// Mitsubishi GX Works2 project: 21_01   PLC: FX3G

// global labels: Global1
VAR_GLOBAL
  switch_check_start AT X007 : BOOL;
  finish_packing AT Y002 : BOOL;
  Not_sufficnt_stuff AT M1 : BOOL;
  kashut_container AT D1101 : REAL;
  lata_container AT D1201 : REAL;
  shmarim_container AT D1202 : REAL;
END_VAR
VAR_GLOBAL CONSTANT
  con120 : REAL := 120;
  cons6 : REAL := 6;
  cons54 : REAL := 54;
END_VAR
VAR_GLOBAL
  Y_7 AT Y007 : BOOL;
  X_11 AT X011 : BOOL;
  Urgent_Shut AT X011 : BOOL;
  start_cook AT X001 : BOOL;
  analog_input AT D8281 : INT;
END_VAR
VAR_GLOBAL CONSTANT
  con400 : INT := 400;
END_VAR
VAR_GLOBAL
  correct_analog AT D1111 : INT;
END_VAR
VAR_GLOBAL CONSTANT
  cons_5 : INT := 5;
END_VAR
VAR_GLOBAL
  what_is_it AT M12 : BOOL;
  NO AT M12 : BOOL;
  Yes_Lager AT M12 : BOOL;
END_VAR
VAR_GLOBAL CONSTANT
  cons_120 : REAL := 120;
  cons_6 : REAL := 6;
END_VAR
VAR_GLOBAL
  bishul_container AT D1299 : REAL;
END_VAR
VAR_GLOBAL CONSTANT
  cons_54 : REAL := 54;
  cons_150 : REAL := 150;
  cons_12 : REAL := 12;
  cons_60 : REAL := 60;
END_VAR
VAR_GLOBAL
  Y_3 AT Y003 : BOOL;
  M_12 AT M12 : BOOL;
  M_13 AT M13 : BOOL;
  Yes_philenzer AT M12 : BOOL;
END_VAR
VAR_GLOBAL CONSTANT
  cons_0 : REAL;
  cons_126 : REAL := 126;
END_VAR
VAR_GLOBAL
  M_17 AT M17 : BOOL;
  cooke_timer AT TC5 : BOOL;
END_VAR
VAR_GLOBAL CONSTANT
  sec_4 : INT := 40;
END_VAR
VAR_GLOBAL
  stop_cooke AT TS5 : BOOL;
  stop_cook AT TS5 : BOOL;
  lamp1_off AT Y001 : BOOL;
  X_5 AT X005 : BOOL;
  tsisa_container AT D1301 : REAL;
  end_cook_lam AT M3 : BOOL;
  BE_counter AT TC2 : BOOL;
END_VAR
VAR_GLOBAL CONSTANT
  Four_sec : INT := 40;
END_VAR
VAR_GLOBAL
  BE_OFF AT TS2 : BOOL;
  Helo_Lamp AT M0 : BOOL;
  Timer_1 AT TC3 : BOOL;
END_VAR
VAR_GLOBAL CONSTANT
  One_sec : INT := 10;
END_VAR
VAR_GLOBAL
  end_timer1 AT TS3 : BOOL;
  Lamp_1 AT Y004 : BOOL;
  Lamp_4 AT Y004 : BOOL;
  Timer_2 AT TC4 : BOOL;
  end_Timer2 AT TS4 : BOOL;
  lamp3 AT Y003 : BOOL;
  lamp0 AT Y003 : BOOL;
  lamlam AT X003 : BOOL;
END_VAR
VAR_GLOBAL CONSTANT
  cons0 : REAL;
END_VAR
VAR_GLOBAL
  BD_counter AT TC6 : BOOL;
  BD_OFF AT TS6 : BOOL;
END_VAR
VAR_GLOBAL CONSTANT
  Three_sec : INT := 30;
END_VAR
VAR_GLOBAL
  Timer_3 AT TC7 : BOOL;
  end_timer3 AT TS7 : BOOL;
  Timer_4 AT TC8 : BOOL;
  end_Timer4 AT TS8 : BOOL;
  Helo_Lamp2 AT M2 : BOOL;
  start_pac AT X002 : BOOL;
  end_tsisa AT M5 : BOOL;
  Nora AT Y006 : BOOL;
  cc1_counter AT CC1 : BOOL;
END_VAR
VAR_GLOBAL CONSTANT
  count1 : WORD := K1;
END_VAR
VAR_GLOBAL
  cc6_counter AT CC6 : BOOL;
END_VAR
VAR_GLOBAL CONSTANT
  count6 : WORD := K6;
END_VAR
VAR_GLOBAL
  cs1 AT CS1 : BOOL;
  cs6 AT CS6 : BOOL;
  y_2 AT Y002 : BOOL;
  x_0 AT X000 : BOOL;
  ready_container AT D1401 : REAL;
END_VAR
VAR_GLOBAL CONSTANT
  add_abeer : REAL := 6;
  add_shishia : REAL := 1;
  con_40 : REAL := 40;
END_VAR
VAR_GLOBAL
  D_4001 AT D4001 : REAL;
  analog_output AT D8282 : INT;
  D_4000 AT D4000 : REAL;
  break AT M14 : BOOL;
END_VAR
VAR_GLOBAL CONSTANT
  mul_1 : REAL := 1;
END_VAR

// task Task_01 (event TRUE, interval 0, priority 31): POU_01

PROGRAM POU_01
(* structured ladder/FBD written out as ST: instructions are called as NAME(EN, inputs, outputs); _pN, _eN, _tN stand for wires *)
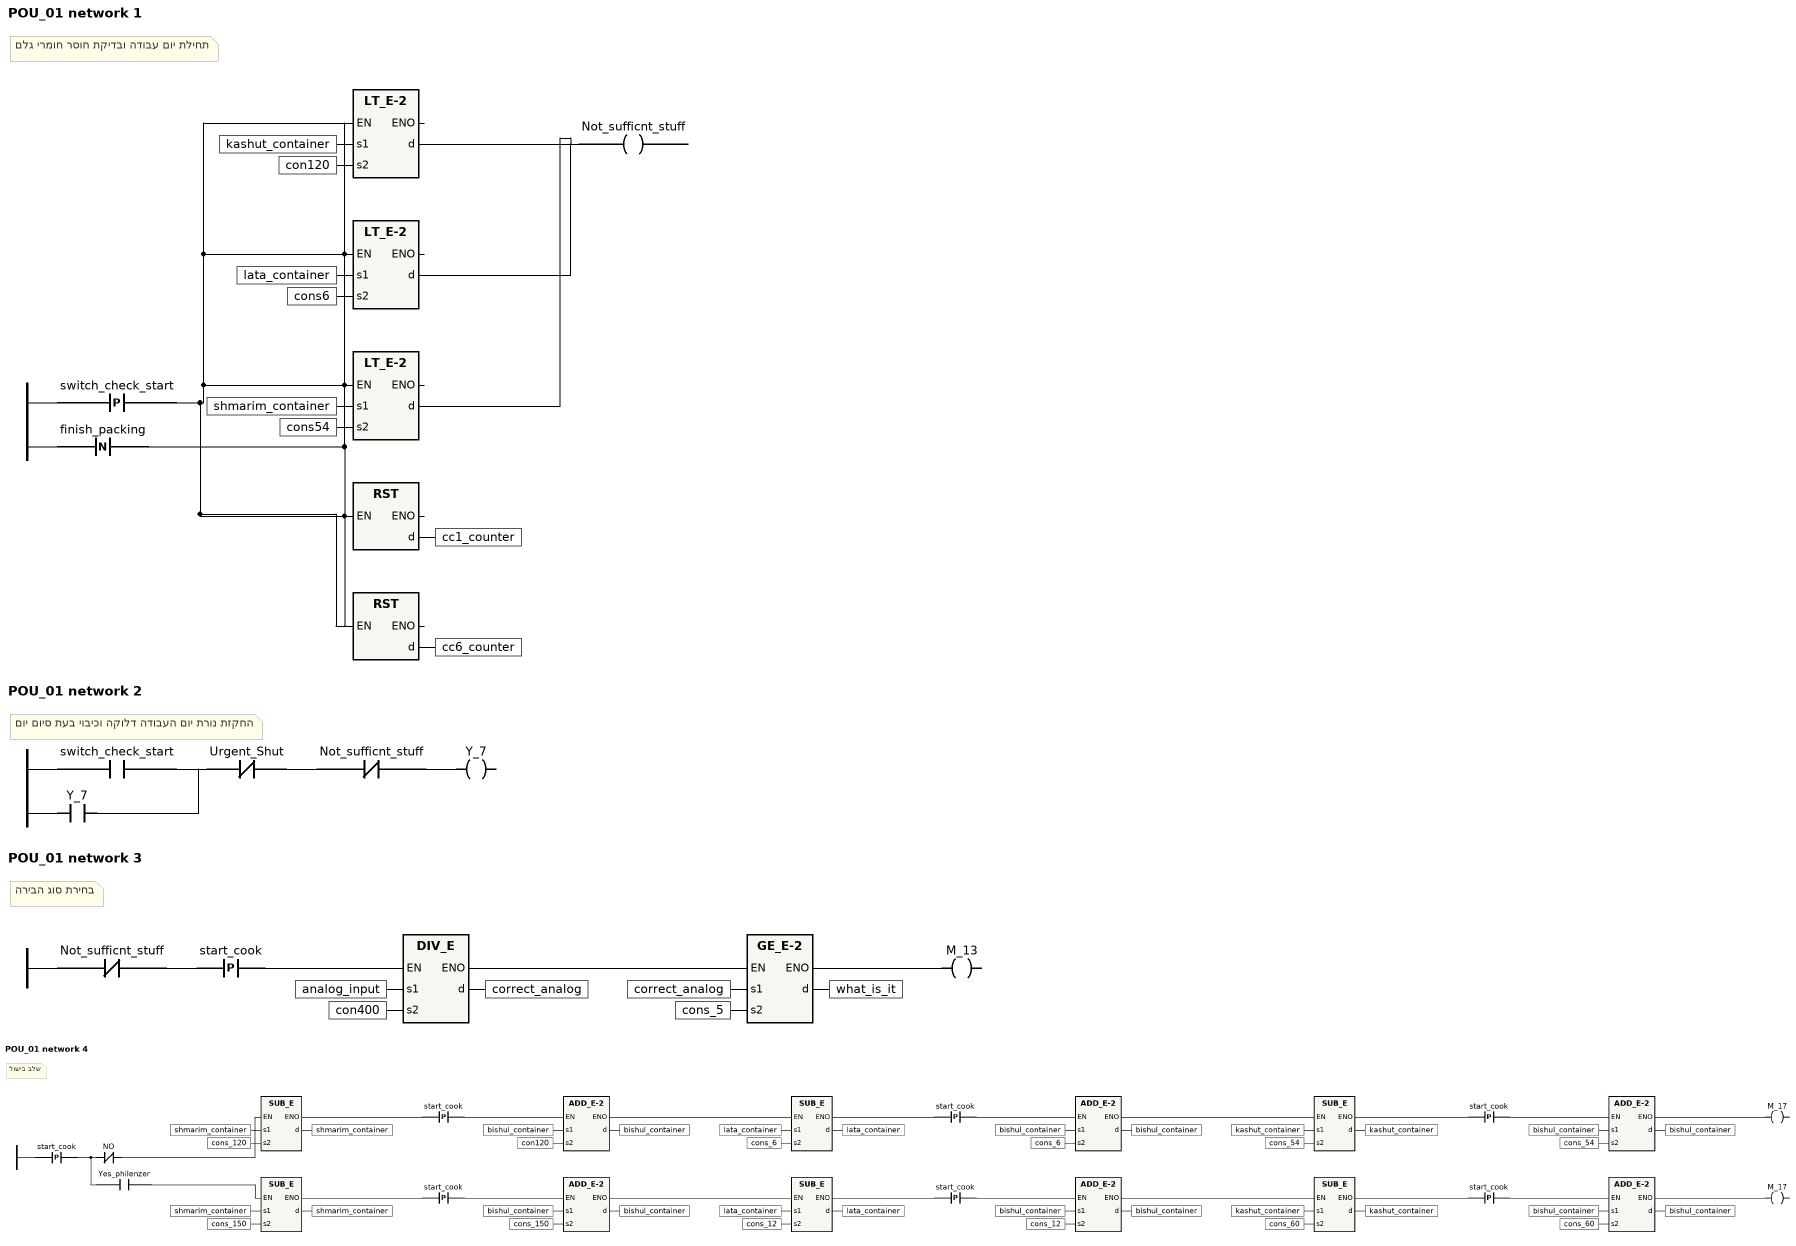
(* network 1 *)
(* תחילת יום עבודה ובדיקת חוסר חומרי גלם *)
_p1 := LDP(TRUE, switch_check_start) OR LDF(TRUE, finish_packing);
LT_E(_p1, kashut_container, con120, _t2);
LT_E(_p1, lata_container, cons6, _t3);
LT_E(_p1, shmarim_container, cons54, _t4);
Not_sufficnt_stuff := _t2 OR _t3 OR _t4;
RST(_p1, cc1_counter);
RST(_p1, cc6_counter);
(* network 2 *)
(* החקזת נורת יום העבודה דלוקה וכיבוי בעת סיום יום *)
Y_7 := ((switch_check_start OR Y_7) AND NOT Urgent_Shut) AND NOT Not_sufficnt_stuff;
(* network 3 *)
(* בחירת סוג הבירה *)
_e1 := DIV_E(NOT Not_sufficnt_stuff AND LDP(TRUE, start_cook), analog_input, con400, correct_analog);
_e2 := GE_E(_e1, correct_analog, cons_5, what_is_it);
M_13 := _e2;
(* network 4 *)
(* שלב בישול *)
_p1 := LDP(TRUE, start_cook);
_e2 := SUB_E(_p1 AND NOT NO, shmarim_container, cons_120, shmarim_container);
_e3 := ADD_E(_e2 AND LDP(TRUE, start_cook), bishul_container, con120, bishul_container);
_e4 := SUB_E(_e3, lata_container, cons_6, lata_container);
_e5 := ADD_E(_e4 AND LDP(TRUE, start_cook), bishul_container, cons_6, bishul_container);
_e6 := SUB_E(_e5, kashut_container, cons_54, kashut_container);
_e7 := ADD_E(_e6 AND LDP(TRUE, start_cook), bishul_container, cons_54, bishul_container);
M_17 := _e7;
_e8 := SUB_E(_p1 AND Yes_philenzer, shmarim_container, cons_150, shmarim_container);
_e9 := ADD_E(_e8 AND LDP(TRUE, start_cook), bishul_container, cons_150, bishul_container);
_e10 := SUB_E(_e9, lata_container, cons_12, lata_container);
_e11 := ADD_E(_e10 AND LDP(TRUE, start_cook), bishul_container, cons_12, bishul_container);
_e12 := SUB_E(_e11, kashut_container, cons_60, kashut_container);
_e13 := ADD_E(_e12 AND LDP(TRUE, start_cook), bishul_container, cons_60, bishul_container);
M_17 := _e13;
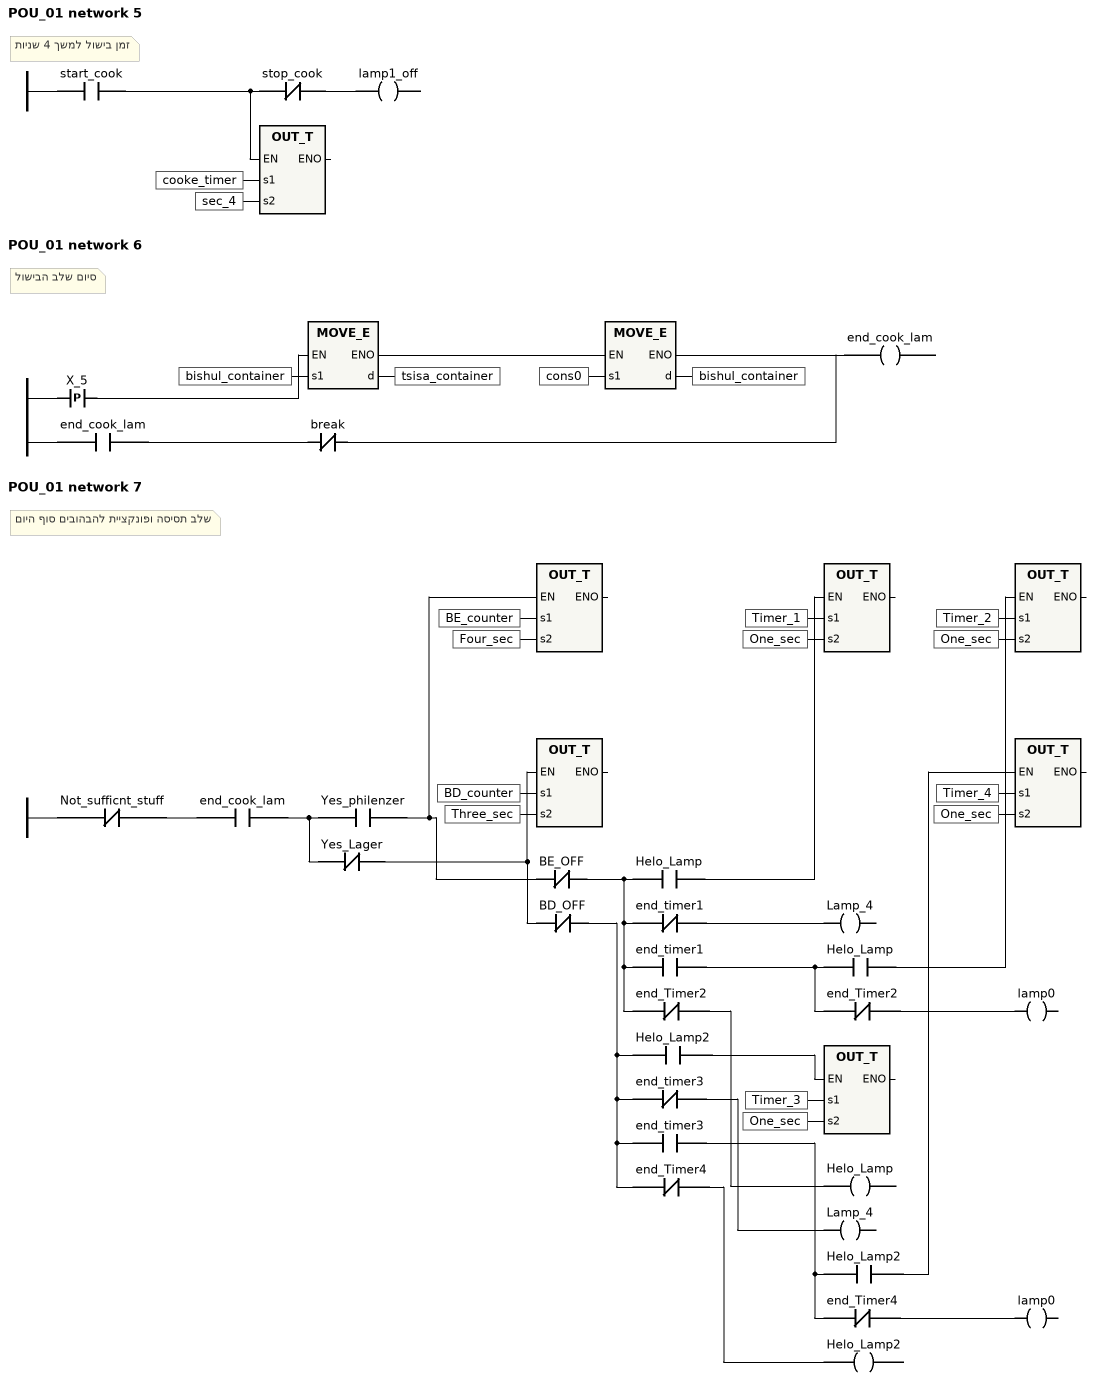
(* network 5 *)
(* זמן בישול למשך 4 שניות *)
lamp1_off := start_cook AND NOT stop_cook;
OUT_T(start_cook, cooke_timer, sec_4);
(* network 6 *)
(* סיום שלב הבישול *)
_e1 := MOVE_E(LDP(TRUE, X_5), bishul_container, tsisa_container);
_e2 := MOVE_E(_e1, cons0, bishul_container);
end_cook_lam := _e2 OR (end_cook_lam AND NOT break);
(* network 7 *)
(* שלב תסיסה ופונקציית להבהובים סוף היום *)
_p1 := NOT Not_sufficnt_stuff AND end_cook_lam;
_p2 := _p1 AND Yes_philenzer;
OUT_T(_p2, BE_counter, Four_sec);
_p3 := _p2 AND NOT BE_OFF;
OUT_T(_p3 AND Helo_Lamp, Timer_1, One_sec);
Lamp_4 := _p3 AND NOT end_timer1;
_p4 := _p3 AND end_timer1;
OUT_T(_p4 AND Helo_Lamp, Timer_2, One_sec);
lamp0 := _p4 AND NOT end_Timer2;
Helo_Lamp := _p3 AND NOT end_Timer2;
_p5 := _p1 AND NOT Yes_Lager;
OUT_T(_p5, BD_counter, Three_sec);
_p6 := _p5 AND NOT BD_OFF;
OUT_T(_p6 AND Helo_Lamp2, Timer_3, One_sec);
Lamp_4 := _p6 AND NOT end_timer3;
_p7 := _p6 AND end_timer3;
OUT_T(_p7 AND Helo_Lamp2, Timer_4, One_sec);
lamp0 := _p7 AND NOT end_Timer4;
Helo_Lamp2 := _p6 AND NOT end_Timer4;
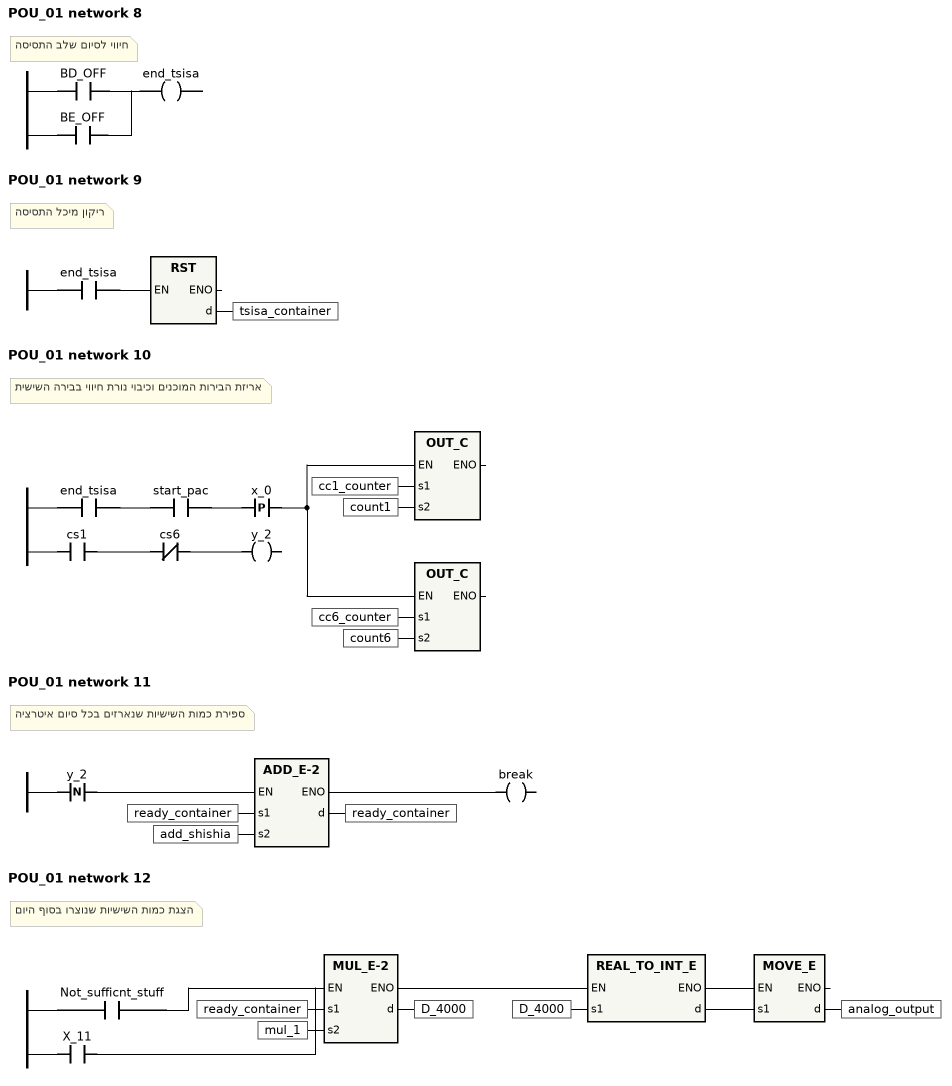
(* network 8 *)
(* חיווי לסיום שלב התסיסה *)
end_tsisa := BD_OFF OR BE_OFF;
(* network 9 *)
(* ריקון מיכל התסיסה *)
RST(end_tsisa, tsisa_container);
(* network 10 *)
(* אריזת הבירות המוכנים וכיבוי נורת חיווי בבירה השישית *)
_p1 := end_tsisa AND start_pac AND LDP(TRUE, x_0);
OUT_C(_p1, cc1_counter, count1);
OUT_C(_p1, cc6_counter, count6);
y_2 := cs1 AND NOT cs6;
(* network 11 *)
(* ספירת כמות השישיות שנארזים בכל סיום איטרציה *)
_e1 := ADD_E(LDF(TRUE, y_2), ready_container, add_shishia, ready_container);
break := _e1;
(* network 12 *)
(* הצגת כמות השישיות שנוצרו בסוף היום *)
_e1 := MUL_E(Not_sufficnt_stuff OR X_11, ready_container, mul_1, D_4000);
_e3 := REAL_TO_INT_E(_e1, D_4000, _t2);
MOVE_E(_e3, _t2, analog_output);
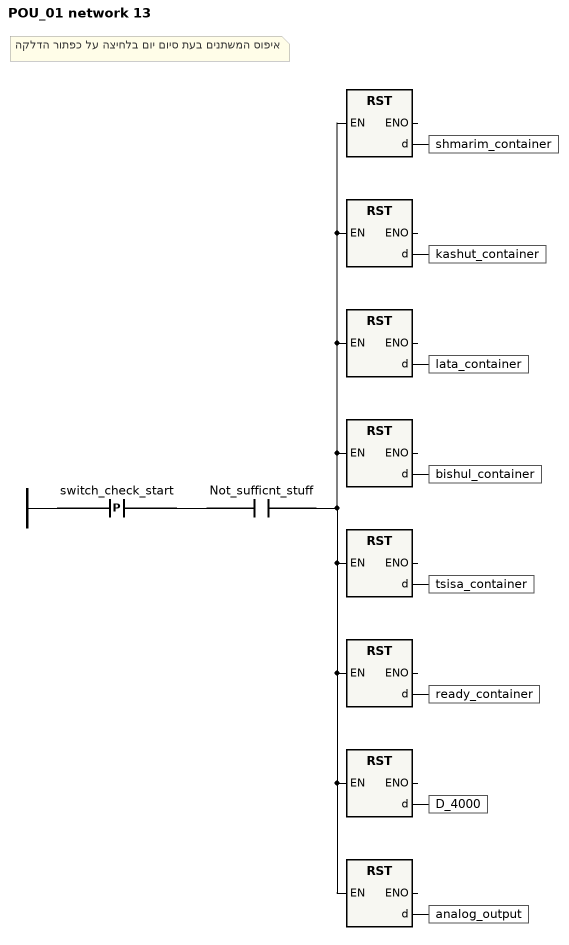
(* network 13 *)
(* איפוס המשתנים בעת סיום יום בלחיצה על כפתור הדלקה *)
_p1 := LDP(TRUE, switch_check_start) AND Not_sufficnt_stuff;
RST(_p1, shmarim_container);
RST(_p1, kashut_container);
RST(_p1, lata_container);
RST(_p1, bishul_container);
RST(_p1, tsisa_container);
RST(_p1, ready_container);
RST(_p1, D_4000);
RST(_p1, analog_output);
END_PROGRAM
